// TIA Portal V18 export
// export: Created 2023-08-15T09:22:34.368735Z, ExportSetting WithDefaults, DisplayName Totally Integrated Automation Portal, DisplayVersion V18 Update 2, DisplayName TIA Portal Openness, DisplayVersion V18 Update 2, DisplayName TIA Portal Version Control Interface, DisplayVersion V18, DisplayName SINAMICS Startdrive Advanced, DisplayVersion V18, DisplayName SINAMICS Startdrive G130, G150, S120, S150, SINAMICS MV, S210, DisplayVersion V18, DisplayName SINAMICS Startdrive G110M, G120, G120C, G120D, G120P, G115D, DisplayVersion V18, DisplayName STEP 7 Professional, DisplayVersion V18 Update 2, DisplayName STEP 7 Safety, DisplayVersion V18, DisplayName WinCC Advanced / Unified PC, DisplayVersion V18 Update 2
ORGANIZATION_BLOCK "Drives"   // OB123, LAD, ProgramCycle
TITLE = "Main Program Sweep (Cycle)"
{ S7_Optimized_Access := 'TRUE' }
VERSION : 0.1
// stored: AutoNumber true, IsIECCheckEnabled false, SetENOAutomatically false
   VAR_INPUT
      Initial_Call : Bool;   // Initial call of this OB
      Remanence : Bool;   // =True, if remanent data are available
   END_VAR
BEGIN

REGION Network 1
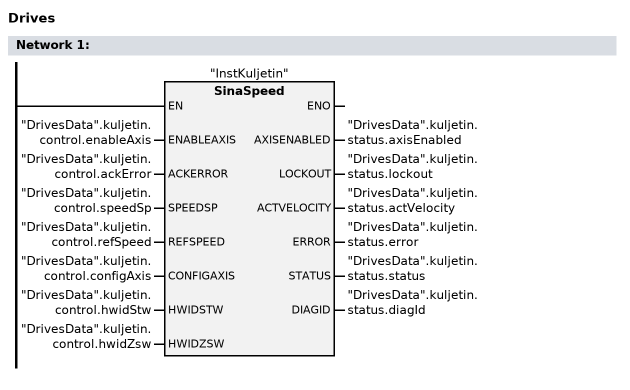
   RUNG wire#powerrail
      "InstKuljetin".SinaSpeed(EnableAxis := "DrivesData".kuljetin.control.enableAxis, AckError := "DrivesData".kuljetin.control.ackError, SpeedSp := "DrivesData".kuljetin.control.speedSp, RefSpeed := "DrivesData".kuljetin.control.refSpeed, ConfigAxis := "DrivesData".kuljetin.control.configAxis, HWIDSTW := "DrivesData".kuljetin.control.hwidStw, HWIDZSW := "DrivesData".kuljetin.control.hwidZsw, AxisEnabled => "DrivesData".kuljetin.status.axisEnabled, Lockout => "DrivesData".kuljetin.status.lockout, ActVelocity => "DrivesData".kuljetin.status.actVelocity, Error => "DrivesData".kuljetin.status.error, Status => "DrivesData".kuljetin.status.status, DiagId => "DrivesData".kuljetin.status.diagId)
   END_RUNG
   // the same network as SCL:
   "InstKuljetin"(EnableAxis := "DrivesData".kuljetin.control.enableAxis,   // SinaSpeed
                  AckError := "DrivesData".kuljetin.control.ackError,
                  SpeedSp := "DrivesData".kuljetin.control.speedSp,
                  RefSpeed := "DrivesData".kuljetin.control.refSpeed,
                  ConfigAxis := "DrivesData".kuljetin.control.configAxis,
                  HWIDSTW := "DrivesData".kuljetin.control.hwidStw,
                  HWIDZSW := "DrivesData".kuljetin.control.hwidZsw,
                  AxisEnabled => "DrivesData".kuljetin.status.axisEnabled,
                  Lockout => "DrivesData".kuljetin.status.lockout,
                  ActVelocity => "DrivesData".kuljetin.status.actVelocity,
                  Error => "DrivesData".kuljetin.status.error,
                  Status => "DrivesData".kuljetin.status.status,
                  DiagId => "DrivesData".kuljetin.status.diagId);
END_REGION
END_ORGANIZATION_BLOCK
